FUNCTION_BLOCK Dispositivo
VAR
	_conexion : I_Conexion;
END_VAR

METHOD establecerConexion 
VAR_INPUT
END_VAR
_conexion.EstablecerConexion();
END_METHOD

METHOD FB_init : BOOL
VAR_INPUT
	bInitRetains : BOOL; // if TRUE, the retain variables are initialized (warm start / cold start)
	bInCopyCode : BOOL;  // if TRUE, the instance afterwards gets moved into the copy code (online change)
	conexion : I_Conexion;
END_VAR
THIS^._conexion := conexion;
END_METHOD

END_FUNCTION_BLOCK

(* stored: Version 1.1.0.1, ProductVersion 3.1.4024.12
   POU Dispositivo: Id {473cbefa-2816-40a9-8a53-8ae3f5bd6201}, SpecialFunc None
   Method establecerConexion: Id {d8dd92d6-a6fc-45c7-922e-c50c39ef05e5}
   Method FB_init: Id {f22fe6c4-dede-48bc-a7d2-e9cefd03731f} *)
